PROGRAM PRG_PID_CALL
VAR
END_VAR

END_PROGRAM

(* stored: Version 1.1.0.1
   POU PRG_PID_CALL: Id {64db7495-2ded-04e8-2256-4a372158dbbf}, SpecialFunc None *)
